(* IEC 61131-3 sources: SafePLC-Gen-Evaluation/PatchEvaluation-DEXPI-Image-2, 2 files *)

(* ---- io_declarations.st ---- *)
(* ==================================================  *)
(* PLC I/O Variable Declarations — CODESYS 3.5  *)
(* Generated by SafePLC-Gen Multimodal  *)
(* ==================================================  *)

VAR_GLOBAL
    (* --- Analog Inputs ---  *)
    PI_4712.01_Raw               AT %IW0       : INT := 0;    (* PI-4712.01 — Pressure indicator on pump P4712 dischar  *)
    PICSA_4712.02_Raw            AT %IW2       : INT := 0;    (* PICSA-4712.02 — Pressure indicator, controller, switch a  *)
    TICSA_4750.03_Raw            AT %IW4       : INT := 0;    (* TICSA-4750.03 — Temperature indicator, controller, switc  *)
    (* --- Analog Outputs ---  *)
    F.O._Out                     AT %QW0       : INT := 0;    (* F.O. — Control valve with fail-open actuator  *)
    (* --- Digital Inputs ---  *)
    HS_4750.01                   AT %IX0.0     : BOOL := FALSE;    (* HS-4750.01 — Hand switch - manual control station  *)
    (* --- Digital Outputs ---  *)
    SV_104.01                    AT %QX0.0     : BOOL := FALSE;    (* SV-104.01 — Solenoid valve 6 bar, DN 25/50  *)
END_VAR

(* ---- generated_code.st ---- *)
(* Generated by SafePLC-Gen Multimodal — CODESYS 3.5 *)
(* IEC 61131-3 Structured Text *)
(* Date: 2026-04-15T13:08:50.712422 *)

PROGRAM Main_Control

VAR
    (* AT-addressed I/O variables *)
    PI_4712_01_Raw               AT %IW0       : INT := 0;
    PICSA_4712_02_Raw            AT %IW2       : INT := 0;
    TICSA_4750_03_Raw            AT %IW4       : INT := 0;
    F_O_Out                      AT %QW0       : INT := 0;
    HS_4750_01                   AT %IX0.0     : BOOL := FALSE;
    SV_104_01                    AT %QX0.0     : BOOL := FALSE;
END_VAR

VAR
    (* Internal variables *)
    FirstScan                    : BOOL := TRUE;

    (* Scaled process variables *)
    PI_4712_01_Scaled            : REAL := 0.0;
    PICSA_4712_02_Scaled         : REAL := 0.0;
    TICSA_4750_03_Scaled         : REAL := 0.0;

    (* Alarm setpoints *)
    PI_4712_01_HH_SP             : REAL := 150.0;
    PI_4712_01_H_SP              : REAL := 140.0;
    PI_4712_01_L_SP              : REAL := 20.0;
    PI_4712_01_LL_SP             : REAL := 10.0;
    PI_4712_01_Deadband          : REAL := 2.0;

    PICSA_4712_02_HH_SP          : REAL := 160.0;
    PICSA_4712_02_H_SP           : REAL := 150.0;
    PICSA_4712_02_L_SP           : REAL := 25.0;
    PICSA_4712_02_LL_SP          : REAL := 15.0;
    PICSA_4712_02_Deadband       : REAL := 2.0;

    TICSA_4750_03_HH_SP          : REAL := 90.0;
    TICSA_4750_03_H_SP           : REAL := 85.0;
    TICSA_4750_03_L_SP           : REAL := 15.0;
    TICSA_4750_03_LL_SP          : REAL := 10.0;
    TICSA_4750_03_Deadband       : REAL := 1.0;

    (* Alarm booleans *)
    PI_4712_01_HH                : BOOL := FALSE;
    PI_4712_01_H                 : BOOL := FALSE;
    PI_4712_01_L                 : BOOL := FALSE;
    PI_4712_01_LL                : BOOL := FALSE;

    PICSA_4712_02_HH             : BOOL := FALSE;
    PICSA_4712_02_H              : BOOL := FALSE;
    PICSA_4712_02_L              : BOOL := FALSE;
    PICSA_4712_02_LL             : BOOL := FALSE;

    TICSA_4750_03_HH             : BOOL := FALSE;
    TICSA_4750_03_H              : BOOL := FALSE;
    TICSA_4750_03_L              : BOOL := FALSE;
    TICSA_4750_03_LL             : BOOL := FALSE;

    (* Alarm latches *)
    PI_4712_01_HH_Latch          : SR := (S1 := FALSE, R := FALSE);
    PI_4712_01_LL_Latch          : SR := (S1 := FALSE, R := FALSE);
    PICSA_4712_02_HH_Latch       : SR := (S1 := FALSE, R := FALSE);
    PICSA_4712_02_LL_Latch       : SR := (S1 := FALSE, R := FALSE);
    TICSA_4750_03_HH_Latch       : SR := (S1 := FALSE, R := FALSE);
    TICSA_4750_03_LL_Latch       : SR := (S1 := FALSE, R := FALSE);

    (* Acknowledgement inputs *)
    PI_4712_01_HH_Ack            : BOOL := FALSE;
    PI_4712_01_LL_Ack            : BOOL := FALSE;
    PICSA_4712_02_HH_Ack         : BOOL := FALSE;
    PICSA_4712_02_LL_Ack         : BOOL := FALSE;
    TICSA_4750_03_HH_Ack         : BOOL := FALSE;
    TICSA_4750_03_LL_Ack         : BOOL := FALSE;

    (* Control variables *)
    PICSA_4712_02_Setpoint       : REAL := 100.0;
    TICSA_4750_03_Setpoint       : REAL := 50.0;

    (* PID control for PICSA-4712.02 *)
    PICSA_Error                  : REAL := 0.0;
    PICSA_Kp                     : REAL := 1.0;
    PICSA_Ki                     : REAL := 0.1;
    PICSA_Integral               : REAL := 0.0;
    PICSA_Output                 : REAL := 0.0;

    (* On/off control for TICSA-4750.03 *)
    TICSA_Error                  : REAL := 0.0;
    TICSA_Hysteresis             : REAL := 2.0;

    (* System alarm aggregation *)
    System_Alarm                 : BOOL := FALSE;
END_VAR

(* First-scan initialization *)
IF FirstScan THEN
    SV_104_01 := FALSE;
    F_O_Out := 0;
    FirstScan := FALSE;
    RETURN;
END_IF;

(* Scale analog inputs from 4-20mA to engineering units *)
PI_4712_01_Scaled := ((INT_TO_REAL(PI_4712_01_Raw) - 6554.0) / (32767.0 - 6554.0)) * 180.0 + 0.0;
PICSA_4712_02_Scaled := ((INT_TO_REAL(PICSA_4712_02_Raw) - 6554.0) / (32767.0 - 6554.0)) * 200.0 + 0.0;
TICSA_4750_03_Scaled := ((INT_TO_REAL(TICSA_4750_03_Raw) - 6554.0) / (32767.0 - 6554.0)) * 100.0 + 0.0;

(* PI-4712.01 Four-level alarm logic *)
IF PI_4712_01_Scaled >= PI_4712_01_HH_SP THEN
    PI_4712_01_HH_Latch.S1 := TRUE;
ELSIF PI_4712_01_Scaled <= (PI_4712_01_HH_SP - PI_4712_01_Deadband) THEN
    PI_4712_01_HH_Latch.S1 := FALSE;
END_IF;

IF PI_4712_01_HH_Latch.Q1 AND PI_4712_01_HH_Ack AND (PI_4712_01_Scaled <= (PI_4712_01_HH_SP - PI_4712_01_Deadband)) THEN
    PI_4712_01_HH_Latch.R := TRUE;
ELSE
    PI_4712_01_HH_Latch.R := FALSE;
END_IF;

PI_4712_01_HH_Latch();

IF PI_4712_01_Scaled >= PI_4712_01_H_SP THEN
    PI_4712_01_H := TRUE;
ELSIF PI_4712_01_Scaled <= (PI_4712_01_H_SP - PI_4712_01_Deadband) THEN
    PI_4712_01_H := FALSE;
END_IF;

IF PI_4712_01_Scaled <= PI_4712_01_L_SP THEN
    PI_4712_01_L := TRUE;
ELSIF PI_4712_01_Scaled >= (PI_4712_01_L_SP + PI_4712_01_Deadband) THEN
    PI_4712_01_L := FALSE;
END_IF;

IF PI_4712_01_Scaled <= PI_4712_01_LL_SP THEN
    PI_4712_01_LL_Latch.S1 := TRUE;
ELSIF PI_4712_01_Scaled >= (PI_4712_01_LL_SP + PI_4712_01_Deadband) THEN
    PI_4712_01_LL_Latch.S1 := FALSE;
END_IF;

IF PI_4712_01_LL_Latch.Q1 AND PI_4712_01_LL_Ack AND (PI_4712_01_Scaled >= (PI_4712_01_LL_SP + PI_4712_01_Deadband)) THEN
    PI_4712_01_LL_Latch.R := TRUE;
ELSE
    PI_4712_01_LL_Latch.R := FALSE;
END_IF;

PI_4712_01_LL_Latch();

(* PICSA-4712.02 Four-level alarm logic *)
IF PICSA_4712_02_Scaled >= PICSA_4712_02_HH_SP THEN
    PICSA_4712_02_HH_Latch.S1 := TRUE;
ELSIF PICSA_4712_02_Scaled <= (PICSA_4712_02_HH_SP - PICSA_4712_02_Deadband) THEN
    PICSA_4712_02_HH_Latch.S1 := FALSE;
END_IF;

IF PICSA_4712_02_HH_Latch.Q1 AND PICSA_4712_02_HH_Ack AND (PICSA_4712_02_Scaled <= (PICSA_4712_02_HH_SP - PICSA_4712_02_Deadband)) THEN
    PICSA_4712_02_HH_Latch.R := TRUE;
ELSE
    PICSA_4712_02_HH_Latch.R := FALSE;
END_IF;

PICSA_4712_02_HH_Latch();

IF PICSA_4712_02_Scaled >= PICSA_4712_02_H_SP THEN
    PICSA_4712_02_H := TRUE;
ELSIF PICSA_4712_02_Scaled <= (PICSA_4712_02_H_SP - PICSA_4712_02_Deadband) THEN
    PICSA_4712_02_H := FALSE;
END_IF;

IF PICSA_4712_02_Scaled <= PICSA_4712_02_L_SP THEN
    PICSA_4712_02_L := TRUE;
ELSIF PICSA_4712_02_Scaled >= (PICSA_4712_02_L_SP + PICSA_4712_02_Deadband) THEN
    PICSA_4712_02_L := FALSE;
END_IF;

IF PICSA_4712_02_Scaled <= PICSA_4712_02_LL_SP THEN
    PICSA_4712_02_LL_Latch.S1 := TRUE;
ELSIF PICSA_4712_02_Scaled >= (PICSA_4712_02_LL_SP + PICSA_4712_02_Deadband) THEN
    PICSA_4712_02_LL_Latch.S1 := FALSE;
END_IF;

IF PICSA_4712_02_LL_Latch.Q1 AND PICSA_4712_02_LL_Ack AND (PICSA_4712_02_Scaled >= (PICSA_4712_02_LL_SP + PICSA_4712_02_Deadband)) THEN
    PICSA_4712_02_LL_Latch.R := TRUE;
ELSE
    PICSA_4712_02_LL_Latch.R := FALSE;
END_IF;

PICSA_4712_02_LL_Latch();

(* TICSA-4750.03 Four-level alarm logic *)
IF TICSA_4750_03_Scaled >= TICSA_4750_03_HH_SP THEN
    TICSA_4750_03_HH_Latch.S1 := TRUE;
ELSIF TICSA_4750_03_Scaled <= (TICSA_4750_03_HH_SP - TICSA_4750_03_Deadband) THEN
    TICSA_4750_03_HH_Latch.S1 := FALSE;
END_IF;

IF TICSA_4750_03_HH_Latch.Q1 AND TICSA_4750_03_HH_Ack AND (TICSA_4750_03_Scaled <= (TICSA_4750_03_HH_SP - TICSA_4750_03_Deadband)) THEN
    TICSA_4750_03_HH_Latch.R := TRUE;
ELSE
    TICSA_4750_03_HH_Latch.R := FALSE;
END_IF;

TICSA_4750_03_HH_Latch();

IF TICSA_4750_03_Scaled >= TICSA_4750_03_H_SP THEN
    TICSA_4750_03_H := TRUE;
ELSIF TICSA_4750_03_Scaled <= (TICSA_4750_03_H_SP - TICSA_4750_03_Deadband) THEN
    TICSA_4750_03_H := FALSE;
END_IF;

IF TICSA_4750_03_Scaled <= TICSA_4750_03_L_SP THEN
    TICSA_4750_03_L := TRUE;
ELSIF TICSA_4750_03_Scaled >= (TICSA_4750_03_L_SP + TICSA_4750_03_Deadband) THEN
    TICSA_4750_03_L := FALSE;
END_IF;

IF TICSA_4750_03_Scaled <= TICSA_4750_03_LL_SP THEN
    TICSA_4750_03_LL_Latch.S1 := TRUE;
ELSIF TICSA_4750_03_Scaled >= (TICSA_4750_03_LL_SP + TICSA_4750_03_Deadband) THEN
    TICSA_4750_03_LL_Latch.S1 := FALSE;
END_IF;

IF TICSA_4750_03_LL_Latch.Q1 AND TICSA_4750_03_LL_Ack AND (TICSA_4750_03_Scaled >= (TICSA_4750_03_LL_SP + TICSA_4750_03_Deadband)) THEN
    TICSA_4750_03_LL_Latch.R := TRUE;
ELSE
    TICSA_4750_03_LL_Latch.R := FALSE;
END_IF;

TICSA_4750_03_LL_Latch();

(* PI control for PICSA-4712.02 controlling F.O. valve *)
PICSA_Error := PICSA_4712_02_Setpoint - PICSA_4712_02_Scaled;
PICSA_Integral := PICSA_Integral + (PICSA_Ki * PICSA_Error);

IF PICSA_Integral > 100.0 THEN
    PICSA_Integral := 100.0;
ELSIF PICSA_Integral < 0.0 THEN
    PICSA_Integral := 0.0;
END_IF;

PICSA_Output := (PICSA_Kp * PICSA_Error) + PICSA_Integral;

IF PICSA_Output > 100.0 THEN
    PICSA_Output := 100.0;
ELSIF PICSA_Output < 0.0 THEN
    PICSA_Output := 0.0;
END_IF;

(* Convert PI output to raw analog output *)
F_O_Out := REAL_TO_INT(6554.0 + (PICSA_Output / 100.0) * (32767.0 - 6554.0));

(* On/off control for TICSA-4750.03 controlling SV-104.01 *)
TICSA_Error := TICSA_4750_03_Setpoint - TICSA_4750_03_Scaled;

IF HS_4750_01 THEN
    IF TICSA_Error > TICSA_Hysteresis THEN
        SV_104_01 := TRUE;
    ELSIF TICSA_Error < -TICSA_Hysteresis THEN
        SV_104_01 := FALSE;
    END_IF;
ELSE
    SV_104_01 := FALSE;
END_IF;

(* Aggregate all alarm states *)
System_Alarm :=
    PI_4712_01_HH_Latch.Q1 OR PI_4712_01_LL_Latch.Q1 OR
    PI_4712_01_H OR PI_4712_01_L OR
    PICSA_4712_02_HH_Latch.Q1 OR PICSA_4712_02_LL_Latch.Q1 OR
    PICSA_4712_02_H OR PICSA_4712_02_L OR
    TICSA_4750_03_HH_Latch.Q1 OR TICSA_4750_03_LL_Latch.Q1 OR
    TICSA_4750_03_H OR TICSA_4750_03_L;

END_PROGRAM
